% RSLogix 500 project MALETA_NOVA_BAK078.RSS %
PROJECT "UNTITLED"    % processor: MicroLogix 1200 %

PROGRAM FILES
  LAD 2   16 rungs
  LAD 3   11 rungs

DATA FILES
  O0 OUTPUT  6 elements
  I1 INPUT  10 elements
  S2 STATUS  66 elements
  B3 BINARY  1 elements
  T4 TIMER  1 elements
  C5 COUNTER  1 elements
  R6 CONTROL  1 elements
  N7 INTEGER  1 elements

LADDER 2
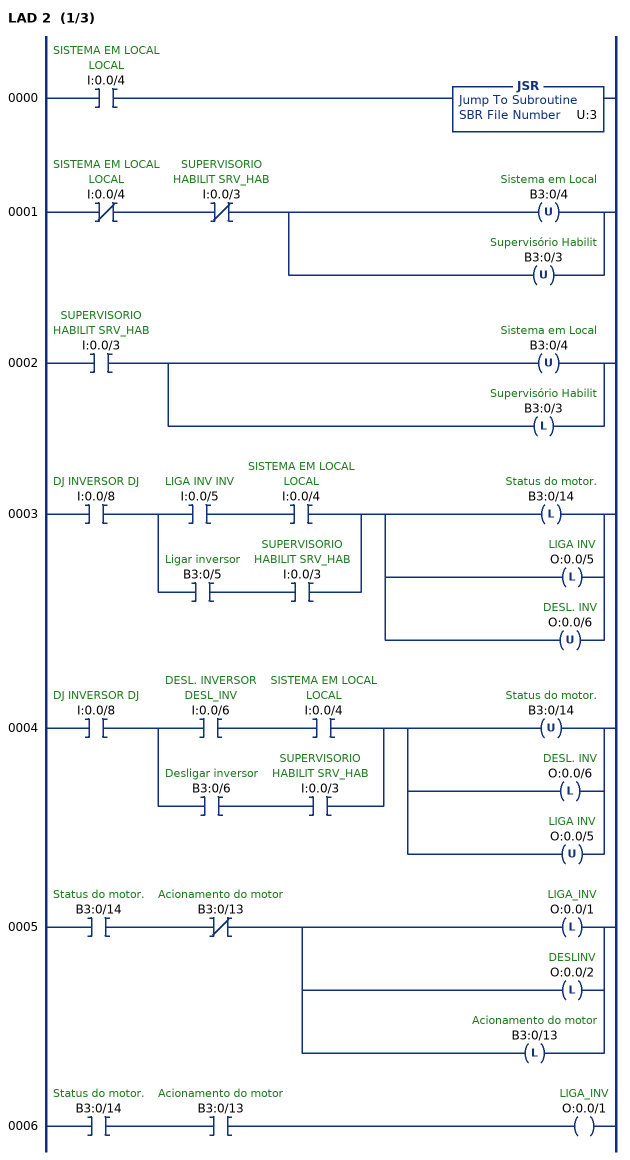
% Rung: 0 %
SOR XIC I:0.0/4 JSR U:3 EOR
%   I:0.0/4  LOCAL  "SISTEMA EM LOCAL" %
% Rung: 1 %  % edit flag set %
SOR XIO I:0.0/4 XIO I:0.0/3 BST OTU B3:0/4 NXB OTU B3:0/3 BND EOR
%   I:0.0/4  LOCAL  "SISTEMA EM LOCAL" %
%   I:0.0/3  SRV_HAB  "SUPERVISORIO HABILIT" %
%   B3:0/4  "Sistema em Local" %
%   B3:0/3  "Supervisório Habilit" %
% Rung: 2 %
SOR XIC I:0.0/3 BST OTU B3:0/4 NXB OTL B3:0/3 BND EOR
%   I:0.0/3  SRV_HAB  "SUPERVISORIO HABILIT" %
%   B3:0/4  "Sistema em Local" %
%   B3:0/3  "Supervisório Habilit" %
% Rung: 3 %
SOR XIC I:0.0/8 BST XIC I:0.0/5 XIC I:0.0/4 NXB XIC B3:0/5 XIC I:0.0/3 BND BST OTL B3:0/14 NXB BST OTL O:0.0/5 NXB OTU O:0.0/6 BND BND EOR
%   I:0.0/8  DJ  "DJ INVERSOR" %
%   I:0.0/5  INV  "LIGA INV" %
%   I:0.0/4  LOCAL  "SISTEMA EM LOCAL" %
%   B3:0/5  "Ligar inversor" %
%   I:0.0/3  SRV_HAB  "SUPERVISORIO HABILIT" %
%   B3:0/14  "Status do motor." %
%   O:0.0/5  "LIGA INV" %
%   O:0.0/6  "DESL. INV" %
% Rung: 4 %
SOR XIC I:0.0/8 BST XIC I:0.0/6 XIC I:0.0/4 NXB XIC B3:0/6 XIC I:0.0/3 BND BST OTU B3:0/14 NXB BST OTL O:0.0/6 NXB OTU O:0.0/5 BND BND EOR
%   I:0.0/8  DJ  "DJ INVERSOR" %
%   I:0.0/6  DESL_INV  "DESL. INVERSOR" %
%   I:0.0/4  LOCAL  "SISTEMA EM LOCAL" %
%   B3:0/6  "Desligar inversor" %
%   I:0.0/3  SRV_HAB  "SUPERVISORIO HABILIT" %
%   B3:0/14  "Status do motor." %
%   O:0.0/6  "DESL. INV" %
%   O:0.0/5  "LIGA INV" %
% Rung: 5 %
SOR XIC B3:0/14 XIO B3:0/13 BST OTL O:0.0/1 NXB BST OTL O:0.0/2 NXB OTL B3:0/13 BND BND EOR
%   B3:0/14  "Status do motor." %
%   B3:0/13  "Acionamento do motor" %
%   O:0.0/1  LIGA_INV %
%   O:0.0/2  DESLINV %
% Rung: 6 %
SOR XIC B3:0/14 XIC B3:0/13 OTE O:0.0/1 EOR
%   B3:0/14  "Status do motor." %
%   B3:0/13  "Acionamento do motor" %
%   O:0.0/1  LIGA_INV %

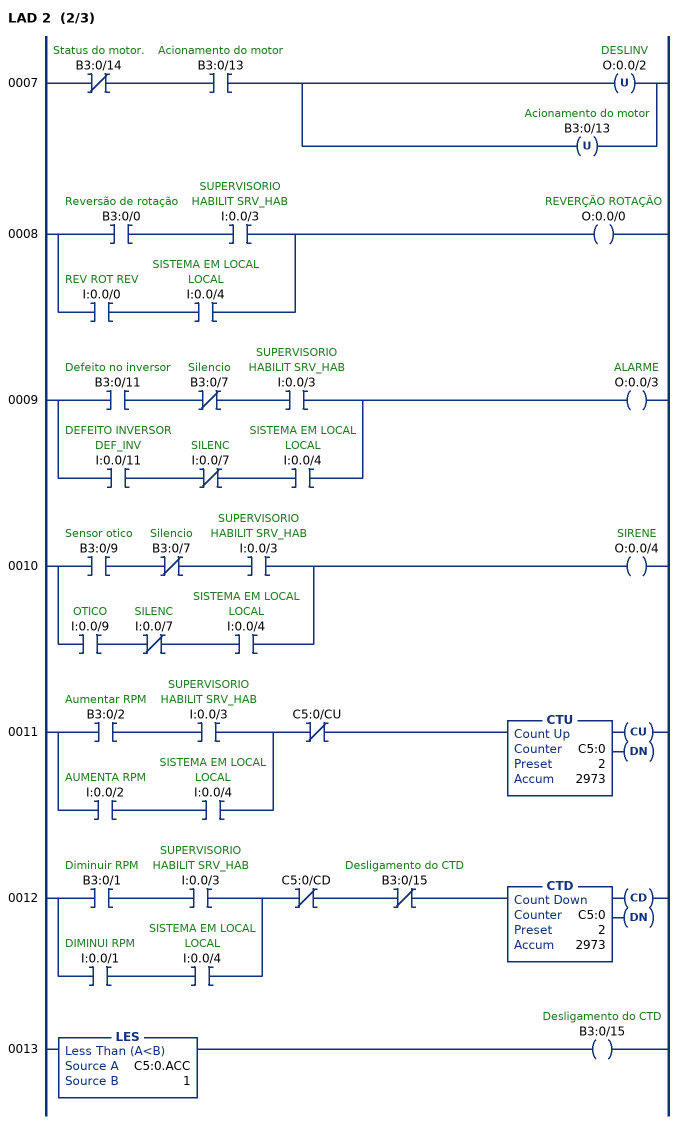
% Rung: 7 %
SOR XIO B3:0/14 XIC B3:0/13 BST OTU O:0.0/2 NXB OTU B3:0/13 BND EOR
%   B3:0/14  "Status do motor." %
%   B3:0/13  "Acionamento do motor" %
%   O:0.0/2  DESLINV %
% Rung: 8 %
SOR BST XIC B3:0/0 XIC I:0.0/3 NXB XIC I:0.0/0 XIC I:0.0/4 BND OTE O:0.0/0 EOR
%   B3:0/0  "Reversão de rotação" %
%   I:0.0/3  SRV_HAB  "SUPERVISORIO HABILIT" %
%   I:0.0/0  REV  "REV ROT" %
%   I:0.0/4  LOCAL  "SISTEMA EM LOCAL" %
%   O:0.0/0  "REVERÇÃO ROTAÇÃO" %
% Rung: 9 %
SOR BST XIC B3:0/11 XIO B3:0/7 XIC I:0.0/3 NXB XIC I:0.0/11 XIO I:0.0/7 XIC I:0.0/4 BND OTE O:0.0/3 EOR
%   B3:0/11  "Defeito no inversor" %
%   B3:0/7  "Silencio" %
%   I:0.0/3  SRV_HAB  "SUPERVISORIO HABILIT" %
%   I:0.0/11  DEF_INV  "DEFEITO INVERSOR" %
%   I:0.0/7  SILENC %
%   I:0.0/4  LOCAL  "SISTEMA EM LOCAL" %
%   O:0.0/3  ALARME %
% Rung: 10 %
SOR BST XIC B3:0/9 XIO B3:0/7 XIC I:0.0/3 NXB XIC I:0.0/9 XIO I:0.0/7 XIC I:0.0/4 BND OTE O:0.0/4 EOR
%   B3:0/9  "Sensor otico" %
%   B3:0/7  "Silencio" %
%   I:0.0/3  SRV_HAB  "SUPERVISORIO HABILIT" %
%   I:0.0/9  OTICO %
%   I:0.0/7  SILENC %
%   I:0.0/4  LOCAL  "SISTEMA EM LOCAL" %
%   O:0.0/4  SIRENE %
% Rung: 11 %
SOR BST XIC B3:0/2 XIC I:0.0/3 NXB XIC I:0.0/2 XIC I:0.0/4 BND XIO C5:0/CU CTU C5:0 2 2973 EOR
%   B3:0/2  "Aumentar RPM" %
%   I:0.0/3  SRV_HAB  "SUPERVISORIO HABILIT" %
%   I:0.0/2  "AUMENTA RPM" %
%   I:0.0/4  LOCAL  "SISTEMA EM LOCAL" %
% Rung: 12 %
SOR BST XIC B3:0/1 XIC I:0.0/3 NXB XIC I:0.0/1 XIC I:0.0/4 BND XIO C5:0/CD XIO B3:0/15 CTD C5:0 2 2973 EOR
%   B3:0/1  "Diminuir RPM" %
%   I:0.0/3  SRV_HAB  "SUPERVISORIO HABILIT" %
%   I:0.0/1  "DIMINUI RPM" %
%   I:0.0/4  LOCAL  "SISTEMA EM LOCAL" %
%   B3:0/15  "Desligamento do CTD" %
% Rung: 13 %
SOR LES C5:0.ACC 1 OTE B3:0/15 EOR
%   B3:0/15  "Desligamento do CTD" %

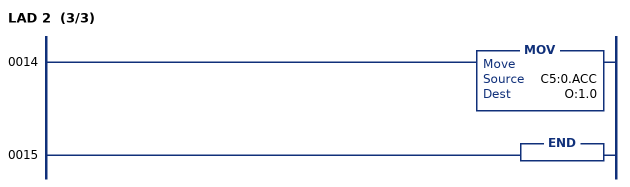
% Rung: 14 %
SOR MOV C5:0.ACC O:1.0 EOR
% Rung: 15 %
SOR END EOR

LADDER 3
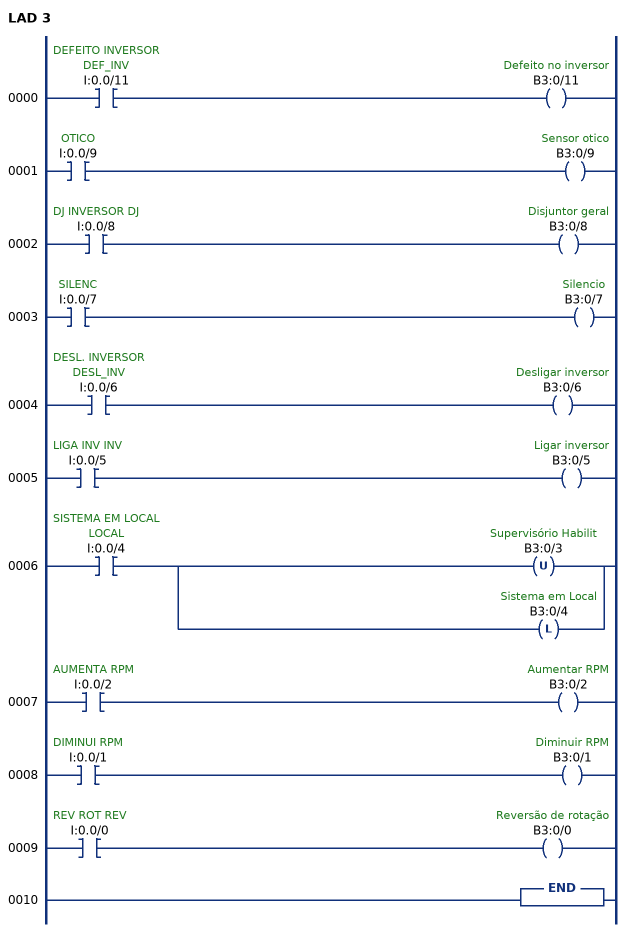
% Rung: 0 %
SOR XIC I:0.0/11 OTE B3:0/11 EOR
%   I:0.0/11  DEF_INV  "DEFEITO INVERSOR" %
%   B3:0/11  "Defeito no inversor" %
% Rung: 1 %
SOR XIC I:0.0/9 OTE B3:0/9 EOR
%   I:0.0/9  OTICO %
%   B3:0/9  "Sensor otico" %
% Rung: 2 %
SOR XIC I:0.0/8 OTE B3:0/8 EOR
%   I:0.0/8  DJ  "DJ INVERSOR" %
%   B3:0/8  "Disjuntor geral" %
% Rung: 3 %
SOR XIC I:0.0/7 OTE B3:0/7 EOR
%   I:0.0/7  SILENC %
%   B3:0/7  "Silencio" %
% Rung: 4 %
SOR XIC I:0.0/6 OTE B3:0/6 EOR
%   I:0.0/6  DESL_INV  "DESL. INVERSOR" %
%   B3:0/6  "Desligar inversor" %
% Rung: 5 %
SOR XIC I:0.0/5 OTE B3:0/5 EOR
%   I:0.0/5  INV  "LIGA INV" %
%   B3:0/5  "Ligar inversor" %
% Rung: 6 %
SOR XIC I:0.0/4 BST OTU B3:0/3 NXB OTL B3:0/4 BND EOR
%   I:0.0/4  LOCAL  "SISTEMA EM LOCAL" %
%   B3:0/3  "Supervisório Habilit" %
%   B3:0/4  "Sistema em Local" %
% Rung: 7 %
SOR XIC I:0.0/2 OTE B3:0/2 EOR
%   I:0.0/2  "AUMENTA RPM" %
%   B3:0/2  "Aumentar RPM" %
% Rung: 8 %
SOR XIC I:0.0/1 OTE B3:0/1 EOR
%   I:0.0/1  "DIMINUI RPM" %
%   B3:0/1  "Diminuir RPM" %
% Rung: 9 %
SOR XIC I:0.0/0 OTE B3:0/0 EOR
%   I:0.0/0  REV  "REV ROT" %
%   B3:0/0  "Reversão de rotação" %
% Rung: 10 %
SOR END EOR

DATA TABLE (non-zero values as saved)
DATA B3
% B3:0 % 0X0110
DATA C5
% .PRE .ACC %
% C5:0 % 2 2973
